RoboDK station: Simulare licenta.rdk

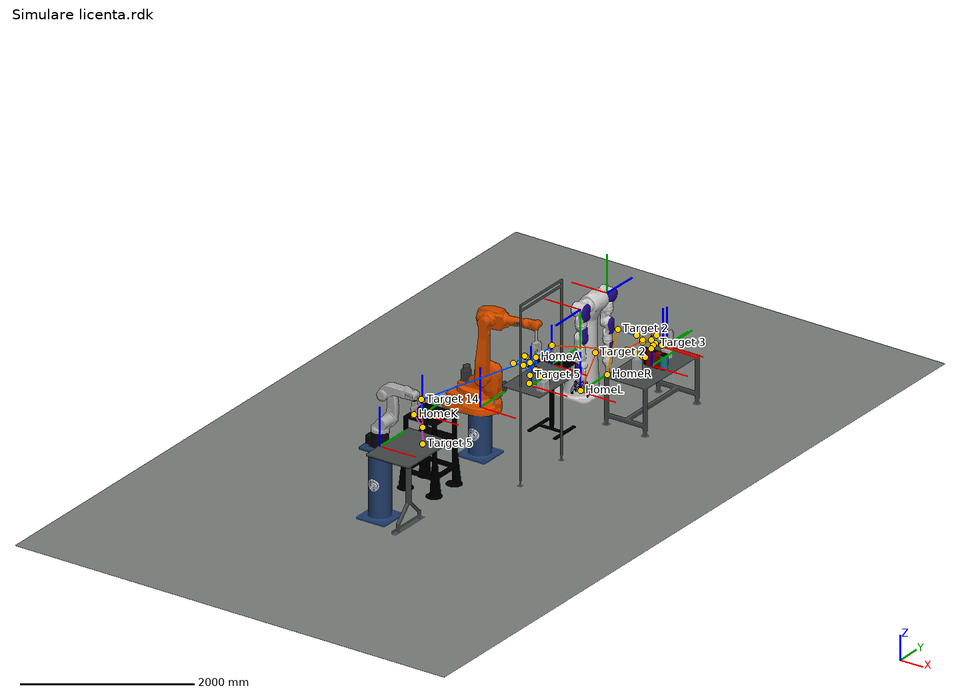
[picture v0: the station drawn from its stored meshes, robots at their saved joint values, targets as dots, program paths as lines]
Station Simulare licenta (saved by RoboDK 5.4.0). Poses are relative to the parent item; angles as X-Y-Z fixed-axis rotations.
  - frame ABB IRB 1600-6/1.45 Base at (0, 0, 600) mm
    - robot ABB IRB 1600-6/1.45: 6 axes, payload 6 kg, reach 1450 mm, repeatability 0.05 mm, weight 250 kg
        modified DH rows (alpha deg, a mm, theta deg, d mm): 0, 0, 0, 486.5; -90, 150, -90, 0; 0, 700, 0, 0; -90, 0, 0, 600; 90, 0, 0, 0; -90, 0, 180, 65
        joint limits [-180, -90, -245, -200, -115, -400] to [180, 120, 65, 200, 115, 400]; home [0, 0, 0, 0, 0, 0]; saved at [3.661, 0.324, -5.471, 0, 95.147, 3.661]
      - tool SCHUNK_0371103_PGN_plus_125_1__000, TCP at (0, 0, 350) mm, size 60 x 151.3 x 378 mm, geometry from SCHUNK_0371103_PGN_plus_125_1__000.stp
    - target HomeA (Cartesian target) at (750, 47.99, 825.32) mm, rotated rx 180 ry 0 rz -180 deg; joints [3.661, 0.324, -5.471, 0, 95.147, 3.661] of ABB IRB 1600-6/1.45
    - target Target 2 (Cartesian target) at (287.69, 1007.38, 456.93) mm, rotated rx 180 ry 0 rz -180 deg; joints [74.062, 29.214, -7.135, 0, 67.921, 74.062] of ABB IRB 1600-6/1.45
    - target Target 3 (Cartesian target) at (287.69, 1001.26, 332.84) mm, rotated rx 180 ry 0 rz -180 deg; joints [73.969, 33.457, -0.924, 0, 57.468, 73.969] of ABB IRB 1600-6/1.45
    - target Target 4 (Cartesian target) at (750, 47.99, 674.68) mm, rotated rx 180 ry 0 rz -180 deg; joints [3.661, 0.768, 8.512, 0, 80.72, 3.661] of ABB IRB 1600-6/1.45
    - target Target 5 (Cartesian target) at (852.72, -221.7, 732.38) mm, rotated rx 180 ry 89.49 rz 180 deg; joints [-26.861, -4.787, 53.092, 145.616, 53.133, -157.935] of ABB IRB 1600-6/1.45
    - target Target 6 (Cartesian target) at (849.34, -221.7, 627.88) mm, rotated rx 180 ry 89.49 rz 180 deg; joints [-27.04, 7.763, 58.334, 150.719, 68.35, -168.569] of ABB IRB 1600-6/1.45
    - target Target 7 (Cartesian target) at (750, -199.45, 825.32) mm, rotated rx 180 ry 0 rz -180 deg; joints [-14.893, 2.337, -7.538, 0, 95.202, -14.893] of ABB IRB 1600-6/1.45
    - target Target 8 (Cartesian target) at (854.13, -221.7, 892.62) mm, rotated rx 180 ry 89.5 rz 180 deg; joints [-26.786, -16.432, 42.285, 130.237, 36.18, -136.606] of ABB IRB 1600-6/1.45
    - target Target 9 (Cartesian target) at (925.55, -221.7, 818.94) mm, rotated rx 180 ry 44.11 rz -180 deg; joints [-19.198, -5.919, 12.219, 19.634, 42.934, -28.675] of ABB IRB 1600-6/1.45
    - target Target 10 (Cartesian target) at (925.55, -221.7, 818.94) mm, rotated rx 180 ry 89.61 rz 180 deg; joints [-23.472, -5.96, 42.941, 143.905, 42.537, -151.925] of ABB IRB 1600-6/1.45
    - target Target 11 (Cartesian target) at (623.92, -221.7, 821.01) mm, rotated rx 180 ry 89.61 rz 180 deg; joints [-46.699, -34.358, 57.99, 110.262, 50.873, -120.743] of ABB IRB 1600-6/1.45
    - target Target 12 (Cartesian target) at (636.73, 6.14, 820.92) mm, rotated rx -90.46 ry 31.14 rz -90.24 deg; joints [1.585, -46.941, 60.499, 6.927, -13.259, -65.588] of ABB IRB 1600-6/1.45
    - target Target 13 (Cartesian target) at (623.92, 5.25, 821.01) mm, rotated rx 180 ry 89.61 rz 180 deg; joints [1.44, -49.033, 60.724, 7.313, -11.39, -7.161] of ABB IRB 1600-6/1.45
    - target Target 14 (Cartesian target) at (-10.54, -1146, 546.53) mm, rotated rx 180 ry 0 rz -180 deg; joints [-90.527, 35.239, -25.964, -180, -80.725, 89.473] of ABB IRB 1600-6/1.45
    - target Target 15 (Cartesian target) at (-10.54, -1146, 387.82) mm, rotated rx 180 ry 0 rz -180 deg; joints [-90.527, 39.032, -16.756, -180, -67.724, 89.473] of ABB IRB 1600-6/1.45
    - target Target 16 (Cartesian target) at (287.69, 1019.67, 456.93) mm, rotated rx 180 ry 0 rz -180 deg; joints [74.244, 30.121, -8.606, 0, 68.485, 74.244] of ABB IRB 1600-6/1.45
    - target Target 17 (Cartesian target) at (985.75, -221.7, 756.85) mm, rotated rx 180 ry 44.11 rz -180 deg; joints [-17.647, -0.333, 13.009, 20.817, 36.422, -29.877] of ABB IRB 1600-6/1.45
    - target Target 18 (Cartesian target) at (985.75, -221.7, 756.85) mm, rotated rx 180 ry 89.15 rz 180 deg; joints [-21.226, 2.977, 41.791, 150.728, 47.764, -159.685] of ABB IRB 1600-6/1.45
    - target Target 19 (Cartesian target) at (985.75, -221.7, 756.85) mm, rotated rx 180 ry 44.11 rz -180 deg; joints [-17.647, -0.333, 13.009, 20.817, 36.422, -29.877] of ABB IRB 1600-6/1.45
    - target Target 20 (Cartesian target) at (985.75, -221.7, 756.85) mm, rotated rx 180 ry 89.15 rz 180 deg; joints [-21.226, 2.977, 41.791, 150.728, 47.764, -159.685] of ABB IRB 1600-6/1.45
  - frame KUKA KR 5 sixx R850 Base at (0, -2000, 900) mm
    - robot KUKA KR 5 sixx R850: 6 axes, payload 5 kg, reach 855 mm, repeatability 0.03 mm, weight 29 kg
        modified DH rows (alpha deg, a mm, theta deg, d mm): 0, 0, 0, 335; -90, 75, 0, 0; 0, 365, -90, 0; -90, 90, 0, 405; 90, 0, 0, 0; -90, 0, 180, 80
        joint limits [-170, -190, -119, -190, -120, -358] to [170, 45, 165, 190, 120, 358]; home [0, -90, 90, 0, 0, 0]; saved at [0, -90, 90, 0, 90, 0]
      - tool 539635_HGP_25_A_B_SSK____asm_0__ZH_, TCP at (0, 0, 170) mm, rotated rx 0 ry 0 rz 180 deg, size 47 x 101 x 197.2 mm, geometry from 539635_HGP_25_A_B_SSK____asm_0__ZH_.stp
    - target HomeK (Cartesian target) at (480, 0, 540) mm, rotated rx -180 ry 0 rz 0 deg; joints [0, -90, 90, 0, 90, 0] of KUKA KR 5 sixx R850
    - target Target 2 (Cartesian target) at (-12.02, 851.6, 253.67) mm, rotated rx 92.47 ry -89.16 rz 180 deg; joints [-90.12, -42.173, 106.544, 2.603, -64.358, -0.286] of KUKA KR 5 sixx R850
    - target Target 4 (Cartesian target) at (577.64, 29.88, 390.74) mm, rotated rx 1.04 ry -89.16 rz 180 deg; joints [-4.42, -93.031, 154.413, -3.815, -62.276, 1.842] of KUKA KR 5 sixx R850
    - target Target 5 (Cartesian target) at (579.54, 29.86, 183.27) mm, rotated rx 1.04 ry -89.16 rz 180 deg; joints [-4.391, -45.31, 147.993, -3.443, -103.501, -0.74] of KUKA KR 5 sixx R850
    - target Target 6 (Cartesian target) at (480, 0, 540) mm, rotated rx -180 ry 0 rz 0 deg; joints [0, -90, 90, 0, 90, 0] of KUKA KR 5 sixx R850
    - target Target 7 (Cartesian target) at (-12.02, 851.6, 253.67) mm, rotated rx 92.47 ry -89.16 rz 180 deg; joints [-90.12, -42.173, 106.544, 2.603, -64.358, -0.286] of KUKA KR 5 sixx R850
    - target Target 7 (Cartesian target) at (-9.43, 851.6, 77.3) mm, rotated rx 92.47 ry -89.16 rz 180 deg; joints [-89.873, -18.515, 95.22, 2.665, -76.682, 0.227] of KUKA KR 5 sixx R850
  - object Pedestal H36in at (0, 0, 0) mm, size 400 x 400 x 914.4 mm, geometry from Pedestal-H36in.sld
  - object masaabb at (0, 0, 0) mm, size 880 x 530 x 2305 mm, geometry from masaabb.stp
  - object Pedestal H24in at (0, 0, 0) mm, size 400 x 400 x 609.6 mm, geometry from Pedestal-H24in.sld
  - object masakuka at (0, 0, 0) mm, size 600 x 850 x 1000 mm, geometry from masakuka.stp
  - object masaintreroboti at (0, -1000, 0) mm, size 600 x 600 x 910 mm, geometry from masaintreroboti.stp
  - frame Frame 6 at (1000, 2000, 610) mm, rotated rx 0.04 ry 0 rz 0 deg
    - object masamotoman at (0, 0, 0) mm, size 640 x 1140 x 615 mm, geometry from masamotoman.stp
    - object suport pahare at (0, -300, 0) mm, rotated rx 0 ry 0 rz 180 deg, size 100 x 100 x 210 mm, geometry from suport pahare.stp
    - object Suport cafea at (0, 0, 0) mm, size 151.2 x 153.3 x 313 mm, geometry from Suport cafea.stl
  - frame Motoman CSDA10F Base at (0, 2000, 0) mm
    - robot Turntable: 1 axes
        modified DH rows (alpha deg, a mm, theta deg, d mm): 0, 0, 0, 0
        base shift (92.5, 0, 0) mm
        joint limits [-200] to [200]; home [0]; saved at [0]
      - frame Right Arm at (100, 265, 1200) mm, rotated rx 90 ry 0 rz -180 deg
        - robot Right CSDA10F (model Motoman CSDA10F): 7 axes, payload 10 kg, reach 720 mm, repeatability 0.6 mm, weight 60 kg
            modified DH rows (alpha deg, a mm, theta deg, d mm): 0, 0, 0, 360; -90, 0, 0, 0; 90, 0, 0, 360; -90, 0, 0, 0; 90, 0, 0, 360; -90, 0, 0, 0; 90, 0, 180, 175
            base shift (0, 0, -360) mm
            joint limits [-180, -110, -170, -135, -180, -110, -180] to [180, 110, 170, 135, 180, 110, 180]; home [90, -90, -90, -130, 0, -60, 90]; saved at [90, -90, 0, 0, 0, 0, 0]
          - tool LEHZ20K2_10_16_0_, TCP at (0, 0, 140) mm, size 81.3 x 34.5 x 159.6 mm, geometry from LEHZ20K2_10_16_0_.stp
        - target HomeR (Cartesian target) at (0, -1035, 0) mm, rotated rx 0 ry 90 rz -90 deg; joints [90, -90, 0, 0, 0, 0, 0] of Right CSDA10F
        - target Target 2 (Cartesian target) at (-146.78, -414.63, 0) mm, rotated rx 0 ry 90 rz -179.5 deg; joints [112.215, -38.164, 0, -103.672, 107.385, 103.215, -36.135] of Right CSDA10F
        - target Target 3 (Cartesian target) at (-649.29, -465.08, 33.19) mm, rotated rx 0 ry 90 rz -179.5 deg; joints [54.13, -49.207, 0, -74.927, 67.545, 60.603, -49.904] of Right CSDA10F
        - target Target 4 (Cartesian target) at (-742.98, -465.91, 33.19) mm, rotated rx 0 ry 90 rz -179.5 deg; joints [47.259, -58.279, 0, -57.417, 67.815, 51.877, -56.553] of Right CSDA10F
        - target Target 5 (Cartesian target) at (-679.15, -330.72, -257.56) mm, rotated rx 0 ry 90 rz -179.5 deg; joints [42.006, -77.982, 0, -79.484, 43.77, 73.322, -15.373] of Right CSDA10F
        - target Target 6 (Cartesian target) at (-821.86, -332.03, -257.56) mm, rotated rx 0 ry 90 rz -179.5 deg; joints [33.009, -88.937, 0, -48.286, 40.963, 55.058, -26.438] of Right CSDA10F
        - target Target 7 (Cartesian target) at (-602.81, -256.65, -278.95) mm, rotated rx 0 ry 90 rz -179.5 deg; joints [41.415, -77.232, 0, -97.556, 41.03, 86.064, -3.419] of Right CSDA10F
        - target Target 8 (Cartesian target) at (-813.1, -258.6, -278.95) mm, rotated rx 0 ry 90 rz -179.5 deg; joints [27.186, -86.811, 0, -59.339, 31.181, 60.152, -16.762] of Right CSDA10F
        - target Target 9 (Cartesian target) at (-812.16, -365.94, -278.95) mm, rotated rx 0 ry 90 rz -179.5 deg; joints [36.148, -94.225, 0, -40.297, 45.644, 54.592, -30.649] of Right CSDA10F
        - target Target 10 (Cartesian target) at (-538.22, -468.56, 212.74) mm, rotated rx -180 ry 62.97 rz 0.5 deg; joints [61.069, -29.073, 0, -54.35, 122.881, 67.492, -110.522] of Right CSDA10F
        - target Target 11 (Cartesian target) at (-766.53, -470.56, 96.28) mm, rotated rx 180 ry 62.97 rz 0.5 deg; joints [43.929, -64.378, 0, -12.171, 134.051, 58.432, -128.308] of Right CSDA10F
      - frame Left Arm at (100, -265, 1200) mm, rotated rx -90 ry 0 rz 180 deg
        - robot Left CSDA10F (model Motoman CSDA10F): 7 axes, payload 10 kg, reach 720 mm, repeatability 0.6 mm, weight 60 kg
            modified DH rows (alpha deg, a mm, theta deg, d mm): 0, 0, 0, 360; -90, 0, 0, 0; 90, 0, 0, 360; -90, 0, 0, 0; 90, 0, 0, 360; -90, 0, 0, 0; 90, 0, 180, 175
            base shift (0, 0, -360) mm
            joint limits [-180, -110, -170, -135, -180, -110, -180] to [180, 110, 170, 135, 180, 110, 180]; home [90, 90, -90, -130, 0, -60, 90]; saved at [-90.45, -90.93, 0, 0, 90, 0, -90]
          - tool ROBOTIQ_AGS-001-XXXX_20171116, TCP at (0, 0, 150) mm, size 130.2 x 233.3 x 211.5 mm, geometry from ROBOTIQ_AGS-001-XXXX_20171116.STEP
        - target Target 2 (Cartesian target) at (-208.84, 486.87, 0) mm, rotated rx -90 ry -0.83 rz 89.91 deg; joints [-102.313, -43.74, 0, -92.52, -98.892, 98.414, -47.744] of Left CSDA10F
        - target Target 3 (Cartesian target) at (-669.86, 304.45, 44.19) mm, rotated rx -90 ry -0.83 rz 89.91 deg; joints [-40.579, -35.277, 0, -98.641, -50.903, 56.779, -56.839] of Left CSDA10F
        - target Target 8 (Cartesian target) at (-669.91, 304.4, 43.85) mm, rotated rx 90 ry 0.78 rz -90.09 deg; joints [-40.571, -35.314, 0, -98.646, -50.877, 56.802, 123.169] of Left CSDA10F
        - target Target 5 (Cartesian target) at (-669.9, 307.55, -277.75) mm, rotated rx 90 ry 0.78 rz -90.09 deg; joints [-40.865, -79.854, 0, -81.531, -42.301, 76.009, 101.628] of Left CSDA10F
        - target Target 6 (Cartesian target) at (-669.56, 518.22, -278.86) mm, rotated rx 90 ry 0.78 rz -90.09 deg; joints [-55.594, -96.456, 0, -35.009, -65.533, 64.885, 132.227] of Left CSDA10F
        - target Target 7 (Cartesian target) at (-705.87, 518.26, -277) mm, rotated rx 90 ry 0.78 rz -90.09 deg; joints [-52.949, -101.558, 0, -23.127, -66.682, 60.23, 138.259] of Left CSDA10F
        - target Target 9 (Cartesian target) at (-100.6, 140.55, 710.33) mm, rotated rx 0.4 ry 0.69 rz -90.09 deg; joints [-55.715, 29.267, 0, -106.213, -0.736, 77.293, 145.784] of Left CSDA10F
        - target Target 10 (Cartesian target) at (-110.24, 293.24, 712.34) mm, rotated rx 0.4 ry 0.78 rz -90.09 deg; joints [-70.041, 6.583, 0, -90.245, -0.643, 84.256, 160.014] of Left CSDA10F
        - target Target 11 (Cartesian target) at (-669.91, 304.4, 43.85) mm, rotated rx 90 ry 0.78 rz -90.09 deg; joints [-40.571, -35.314, 0, -98.646, -50.877, 56.802, 123.169] of Left CSDA10F
        - target Target 12 (Cartesian target) at (-785.67, 306.43, 46.88) mm, rotated rx -90 ry 0 rz 90.02 deg; joints [-33.642, -45.628, 0, -79.058, -49.489, 46.813, -51.306] of Left CSDA10F
        - target Target 12 (Cartesian target) at (-785.67, 306.43, 46.88) mm, rotated rx -90 ry 0 rz 90.02 deg; joints [-33.077, -46.752, 0, -76.954, -49.594, 45.821, -50.694] of Left CSDA10F
        - target HomeL (Cartesian target) at (8.13, 1034.83, -16.8) mm, rotated rx -180 ry 89.07 rz -90.45 deg; joints [-90.45, -90.93, 0, 0, 90, 0, -90] of Left CSDA10F
  - program Capula neagra (18 instructions, listed below)
  - program Prog2 (21 instructions, listed below)
  - program Program Motoman (2 instructions, listed below)
  - object masaintremotoabb at (0, 0, 0) mm, size 400 x 400 x 860 mm, geometry from masaintremotoabb.stp
  - program Prog4 (39 instructions, listed below)
  - program Prog5 (12 instructions, listed below)
  - program Prog6 (5 instructions, listed below)
  - frame Frame 7 at (1000, 2000, 610) mm
    - object Nesspreso Essensa Mini v11 at (0, 0, 0) mm, size 330.3 x 112.6 x 205.3 mm, geometry from Nesspreso Essensa Mini v11.iges
  - program Prog7 (6 instructions, listed below)
  - frame Frame 8 at (300, 1000, 830) mm
  - frame Frame 9 at (0, -1145.9, 968.34) mm
    - target Target 3 (Cartesian target) at (-9.43, -2.5, 8.97) mm, rotated rx 92.47 ry -89.16 rz 180 deg; joints [-89.873, -18.515, 95.22, 2.665, -76.682, 0.227] of KUKA KR 5 sixx R850
  - frame Frame 10 at (950, 2300.45, 710) mm
    - object Dolce Gusto capsule at (0, 0, 0) mm, size 53.2 x 54 x 34.7 mm, geometry from Dolce Gusto capsule.STEP
  - frame Frame 11 at (870, -220, 1206) mm
    - object recipient zahar at (160.01, 0.07, -5.93) mm, rotated rx -0.02 ry -0.02 rz 90.02 deg, size 123.8 x 125.4 x 140.2 mm, geometry from recipient zahar.stp
    - object lingurita at (0, 0, 0) mm, size 99.2 x 40.9 x 19 mm, geometry from lingurita.stp
  - object podea at (0, 0, -3) mm, rotated rx 0 ry 0 rz 90 deg, size 10000 x 6000 x 2 mm, geometry from podea.stp
  - Python program mqtt_joints_motoman_left (listed below)
  - Python program mqtt_joints_motoman_right (listed below)
  - Python program mqtt_joints_kuka (listed below)
  - Python program mqtt_joints_abb (listed below)
  - Python program cafea (listed below)
  - program Capsula lapte (19 instructions, listed below)
  - frame Frame 12 at (970, 2350.45, 710) mm
    - object Dolce Gusto capsule at (0, 0, 0) mm, size 53.2 x 54 x 34.7 mm, geometry from Dolce Gusto capsule.STEP
  - program 2 lingurite (47 instructions, listed below)
  - program 3 lingurite (55 instructions, listed below)
  - program neagra2 (6 instructions, listed below)
  - program neagra3 (6 instructions, listed below)
  - program lapte1 (6 instructions, listed below)
  - program lapte2 (6 instructions, listed below)
  - program lapte3 (6 instructions, listed below)
  - object Coffee Cup- at (1000, 1700, 900) mm, size 84.6 x 83.8 x 116.5 mm, geometry from Coffee Cup-.STEP
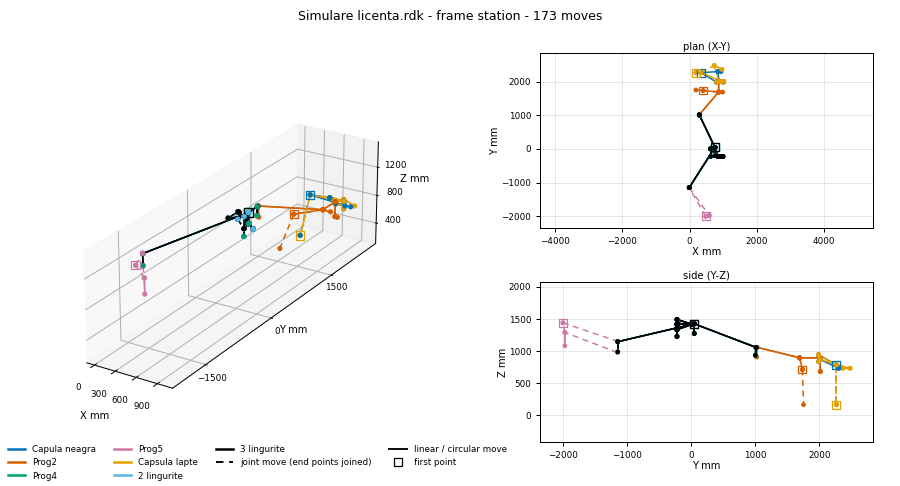
[picture p0: tool path of Simulare licenta.rdk in frame station, 173 of 173 moves have a stored position in this frame; points joined in program order, loops and branches not executed]

--- program Capula neagra (robot Right CSDA10F) ---
  Set Ref.: Right Arm
  MoveJ (Target 2)
  MoveL (Target 3)
  MoveL (Target 4)
  Attach to LEHZ20K2_10_16_0_
  MoveL (Target 3)
  MoveL (Target 5)
  MoveL (Target 6)
  Detach from LEHZ20K2_10_16_0_
  Hide Dolce Gusto capsule
  MoveL (Target 5)
  MoveL (Target 7)
  MoveL (Target 8)
  MoveL (Target 9)
  MoveL (Target 8)
  MoveL (Target 7)
  MoveL (Target 2)
  MoveJ (HomeR)

--- program Prog2 (robot Left CSDA10F) ---
  Set Ref.: Left Arm
  MoveJ (Target 2)
  MoveL (Target 3)
  MoveL (Target 12)
  Attach to ROBOTIQ_AGS-001-XXXX_20171116
  MoveL (Target 3)
  MoveJ (Target 8)
  MoveL (Target 5)
  MoveL (Target 6)
  MoveL (Target 7)
  Pause 10.0 s
  MoveL (Target 6)
  MoveL (Target 5)
  MoveL (Target 8)
  MoveL (Target 9)
  MoveL (Target 10)
  Detach from ROBOTIQ_AGS-001-XXXX_20171116
  MoveL (Target 9)
  MoveL (Target 11)
  MoveJ (Target 2)
  MoveJ (Target 13) -> target HomeL

--- program Program Motoman (robot ABB IRB 1600-6/1.45) ---
  Call Capula neagra
  Call Prog2

--- program Prog4 (robot ABB IRB 1600-6/1.45) ---
  Set Ref.: ABB IRB 1600-6/1.45 Base
  MoveJ (HomeA)
  MoveL (Target 16)
  MoveL (Target 3)
  Attach to SCHUNK_0371103_PGN_plus_125_1__000
  MoveL (Target 2)
  MoveL (HomeA)
  MoveL (Target 4)
  Detach from SCHUNK_0371103_PGN_plus_125_1__000
  MoveL (HomeA)
  MoveL (Target 7)
  MoveJ (Target 5)
  MoveL (Target 6)
  Attach to SCHUNK_0371103_PGN_plus_125_1__000
  MoveL (Target 5)
  MoveL (Target 10)
  MoveJ (Target 9)
  MoveL (Target 19)
  MoveL (Target 20)
  MoveL (Target 10)
  MoveL (Target 8)
  MoveL (Target 13)
  MoveJ (Target 12)
  MoveJ (Target 13)
  MoveL (Target 11)
  MoveL (Target 8)
  MoveL (Target 5)
  MoveL (Target 6)
  Detach from SCHUNK_0371103_PGN_plus_125_1__000
  MoveL (Target 5)
  MoveL (HomeA)
  MoveL (Target 4)
  Attach to SCHUNK_0371103_PGN_plus_125_1__000
  MoveL (HomeA)
  MoveL (Target 14)
  MoveL (Target 15)
  Detach from SCHUNK_0371103_PGN_plus_125_1__000
  MoveL (Target 14)
  MoveL (HomeA)

--- program Prog5 (robot KUKA KR 5 sixx R850) ---
  Set Ref.: KUKA KR 5 sixx R850 Base
  Set Tool: 539635_HGP_25_A_B_SSK____asm_0__ZH_
  MoveJ (Target 6)
  MoveJ (Target 7)
  MoveL (Target 2)
  MoveL (Target 7)
  Attach to 539635_HGP_25_A_B_SSK____asm_0__ZH_
  MoveJ (Target 4)
  MoveL (Target 5)
  Detach from 539635_HGP_25_A_B_SSK____asm_0__ZH_
  MoveL (Target 4)
  MoveJ (HomeK)

--- program Prog6 (robot ABB IRB 1600-6/1.45) ---
  Call Program Motoman
  Call Prog4
  Call Prog5
  Pause 5.0 s
  Call Prog7

--- program Prog7 (robot ABB IRB 1600-6/1.45) ---
  Replace objects
  Replace objects
  Show Dolce Gusto capsule
  Replace objects
  Replace Dolce Gusto capsule
  Show Dolce Gusto capsule

--- Python program mqtt_joints_motoman_left ---
import random

from paho.mqtt import client as mqtt_client

from robodk.robolink import *

RDK = Robolink()
robot  = RDK.Item('Left CSDA10F')

broker = '188.24.48.213'
#broker = '192.168.1.113'
port = 1883
topic = "licenta/jointsmotomanl"
# generate client ID with pub prefix randomly
client_id = f'python-mqtt-{random.randint(0, 100)}'
username = 'basti'
password = 'topsecret'


def connect_mqtt() -> mqtt_client:
    def on_connect(client, userdata, flags, rc):
        if rc == 0:
            print("Connected to MQTT Broker!")
        else:
            print("Failed to connect, return code %d\n", rc)

    client = mqtt_client.Client(client_id)
    client.username_pw_set(username, password)
    client.on_connect = on_connect
    client.connect(broker, port)
    return client

def filtrare (mesaj):
    nc = "{},:'jml "
    for character in nc:
        mesaj = mesaj.replace(character, "")
    j = mesaj.split('"')
    indices = [2, 4, 6, 8, 10, 12, 14]
    print(mesaj)
    extracted_elements = [j[index] for index in indices]
    for i in range(0, len(extracted_elements)):
        extracted_elements[i] = int(extracted_elements[i])
    return extracted_elements

def subscribe(client: mqtt_client):
    def on_message(client, userdata, msg):
        mesaj = msg.payload.decode()
        joints = filtrare(mesaj)
        robot.MoveJ(joints)
    client.subscribe(topic)
    client.on_message = on_message


def run():
    client = connect_mqtt()
    subscribe(client)
    client.loop_forever()


if __name__ == '__main__':
    run()

--- Python program mqtt_joints_motoman_right ---
import random

from paho.mqtt import client as mqtt_client

from robodk.robolink import *

RDK = Robolink()
robot  = RDK.Item('Right CSDA10F')

broker = '188.24.48.213'
#broker = '192.168.1.113'
port = 1883
topic = "licenta/jointsmotomanr"
# generate client ID with pub prefix randomly
client_id = f'python-mqtt-{random.randint(0, 100)}'
username = 'basti'
password = 'topsecret'


def connect_mqtt() -> mqtt_client:
    def on_connect(client, userdata, flags, rc):
        if rc == 0:
            print("Connected to MQTT Broker!")
        else:
            print("Failed to connect, return code %d\n", rc)

    client = mqtt_client.Client(client_id)
    client.username_pw_set(username, password)
    client.on_connect = on_connect
    client.connect(broker, port)
    return client


def filtrare (mesaj):
    nc = "{},:'jmr "
    for character in nc:
        mesaj = mesaj.replace(character, "")
    j = mesaj.split('"')
    indices = [2, 4, 6, 8, 10, 12, 14]
    print(mesaj)
    extracted_elements = [j[index] for index in indices]
    for i in range(0, len(extracted_elements)):
        extracted_elements[i] = int(extracted_elements[i])
    return extracted_elements

def subscribe(client: mqtt_client):
    def on_message(client, userdata, msg):
        mesaj = msg.payload.decode()
        joints = filtrare(mesaj)
        robot.MoveJ(joints)
    client.subscribe(topic)
    client.on_message = on_message


def run():
    client = connect_mqtt()
    subscribe(client)
    client.loop_forever()


if __name__ == '__main__':
    run()

--- Python program mqtt_joints_kuka ---
import random

from paho.mqtt import client as mqtt_client

from robodk.robolink import *

#broker = '192.168.1.113'
broker = '188.24.48.213'
port = 1883
topic = "licenta/jointskuka"
client_id = f'python-mqtt-{random.randint(0, 100)}'
username = 'basti'
password = 'topsecret'
RDK = Robolink()
robot  = RDK.Item('KUKA KR 5 sixx R850')

def connect_mqtt() -> mqtt_client:
    def on_connect(client, userdata, flags, rc):
        if rc == 0:
            print("Connected to MQTT Broker!")
        else:
            print("Failed to connect, return code %d\n", rc)

    client = mqtt_client.Client(client_id)
    client.username_pw_set(username, password)
    client.on_connect = on_connect
    client.connect(broker, port)
    return client


def filtrare(mesaj):
    nc = "{},:'jk "
    for character in nc:
            mesaj = mesaj.replace(character, "")
    j = mesaj.split('"')
    indices = [2, 4, 6, 8, 10, 12]
    print(mesaj)
    extracted_elements = [j[index] for index in indices]
    for i in range(0, len(extracted_elements)):
        extracted_elements[i] = int(extracted_elements[i])
    return extracted_elements

def subscribe(client: mqtt_client):
    def on_message(client, userdata, msg):
        mesaj = msg.payload.decode()
        joints = filtrare(mesaj)
        robot.MoveJ(joints)
    client.subscribe(topic)
    client.on_message = on_message


def run():
    client = connect_mqtt()
    subscribe(client)
    client.loop_forever()


if __name__ == '__main__':
    run()

--- Python program mqtt_joints_abb ---
import random

from paho.mqtt import client as mqtt_client

from robodk.robolink import *

RDK = Robolink()
robot  = RDK.Item('ABB IRB 1600-6/1.45')

broker = '188.24.48.213'
#broker = '192.168.1.113'
port = 1883
topic = "licenta/jointsabb"
# generate client ID with pub prefix randomly
client_id = f'python-mqtt-{random.randint(0, 100)}'
username = 'basti'
password = 'topsecret'


def connect_mqtt() -> mqtt_client:
    def on_connect(client, userdata, flags, rc):
        if rc == 0:
            print("Connected to MQTT Broker!")
        else:
            print("Failed to connect, return code %d\n", rc)

    client = mqtt_client.Client(client_id)
    client.username_pw_set(username, password)
    client.on_connect = on_connect
    client.connect(broker, port)
    return client


def filtrare (mesaj):
    nc = "{},:'ja "
    for character in nc:
        mesaj = mesaj.replace(character, "")
    j = mesaj.split('"')
    indices = [2, 4, 6, 8, 10, 12]
    print(mesaj)
    extracted_elements = [j[index] for index in indices]
    for i in range(0, len(extracted_elements)):
        extracted_elements[i] = int(extracted_elements[i])
    return extracted_elements

def subscribe(client: mqtt_client):
    def on_message(client, userdata, msg):
        mesaj = msg.payload.decode()
        joints = filtrare(mesaj)
        robot.MoveJ(joints)
    client.subscribe(topic)
    client.on_message = on_message


def run():
    client = connect_mqtt()
    subscribe(client)
    client.loop_forever()


if __name__ == '__main__':
    run()

--- Python program cafea ---
import random

from paho.mqtt import client as mqtt_client

from robodk.robolink import *

RDK = Robolink()
robot  = RDK.Item('ABB IRB 1600-6/1.45')
case1 = RDK.Item('Prog6')
case2 = RDK.Item('neagra2')
case3 = RDK.Item('neagra3')
case4 = RDK.Item('lapte1')
case5 = RDK.Item('lapte2')
case6 = RDK.Item('lapte3')

broker = '188.24.48.213'
#broker = '192.168.1.113'
port = 1883
topic = "licenta/cafea"
# generate client ID with pub prefix randomly
client_id = f'python-mqtt-{random.randint(0, 100)}'
username = 'basti'
password = 'topsecret'


def connect_mqtt() -> mqtt_client:
    def on_connect(client, userdata, flags, rc):
        if rc == 0:
            print("Connected to MQTT Broker!")
        else:
            print("Failed to connect, return code %d\n", rc)

    client = mqtt_client.Client(client_id)
    client.username_pw_set(username, password)
    client.on_connect = on_connect
    client.connect(broker, port)
    return client


def caseSelection (mesaj):
    case = int(mesaj)
    print(case)
    if case == 21:
        case1.RunProgram()
        while case1.Busy():
            print("Waiting for the program to complete")
    elif case == 25:
        case2.RunProgram()
        while case2.Busy():
            print("Waiting for the program to complete")
    elif case == 27:
        case3.RunProgram()
        while case3.Busy():
            print("Waiting for the program to complete")
    elif case == 31:
        case4.RunProgram()
        while case4.Busy():
            print("Waiting for the program to complete")
    elif case == 35:
        case5.RunProgram()
        while case5.Busy():
            print("Waiting for the program to complete")
    elif case == 37:
        case6.RunProgram()
        while case6.Busy():
            print("Waiting for the program to complete")

def subscribe(client: mqtt_client):
    def on_message(client, userdata, msg):
        mesaj = msg.payload.decode()
        caseSelection(mesaj)
    client.subscribe(topic)
    client.on_message = on_message


def run():
    client = connect_mqtt()
    subscribe(client)
    client.loop_forever()


if __name__ == '__main__':
    run()

--- program Capsula lapte (robot Right CSDA10F) ---
  Set Ref.: Right Arm
  Set Tool: LEHZ20K2_10_16_0_
  MoveJ (HomeR)
  MoveJ (Target 2)
  MoveJ (Target 10)
  MoveL (Target 11)
  Attach to LEHZ20K2_10_16_0_
  MoveL (Target 10)
  MoveL (Target 5)
  MoveL (Target 6)
  Detach from LEHZ20K2_10_16_0_
  Hide Dolce Gusto capsule
  MoveL (Target 5)
  MoveL (Target 7)
  MoveL (Target 8)
  MoveL (Target 9)
  MoveL (Target 8)
  MoveL (Target 2)
  MoveJ (HomeR)

--- program 2 lingurite (robot ABB IRB 1600-6/1.45) ---
  Set Ref.: ABB IRB 1600-6/1.45 Base
  MoveJ (HomeA)
  MoveL (Target 16)
  MoveL (Target 3)
  Attach to SCHUNK_0371103_PGN_plus_125_1__000
  MoveL (Target 2)
  MoveL (HomeA)
  MoveL (Target 4)
  Detach from SCHUNK_0371103_PGN_plus_125_1__000
  MoveL (HomeA)
  MoveL (Target 7)
  MoveJ (Target 5)
  MoveL (Target 6)
  Attach to SCHUNK_0371103_PGN_plus_125_1__000
  MoveL (Target 5)
  MoveL (Target 10)
  MoveJ (Target 9)
  MoveL (Target 19)
  MoveL (Target 20)
  MoveL (Target 10)
  MoveL (Target 8)
  MoveL (Target 13)
  MoveJ (Target 12)
  MoveJ (Target 13)
  MoveJ (Target 9)
  MoveL (Target 19)
  MoveL (Target 20)
  MoveL (Target 10)
  MoveL (Target 8)
  MoveL (Target 13)
  MoveJ (Target 12)
  MoveJ (Target 13)
  MoveL (Target 11)
  MoveL (Target 8)
  MoveL (Target 5)
  MoveL (Target 6)
  Detach from SCHUNK_0371103_PGN_plus_125_1__000
  MoveL (Target 5)
  MoveL (HomeA)
  MoveL (Target 4)
  Attach to SCHUNK_0371103_PGN_plus_125_1__000
  MoveL (HomeA)
  MoveL (Target 14)
  MoveL (Target 15)
  Detach from SCHUNK_0371103_PGN_plus_125_1__000
  MoveL (Target 14)
  MoveL (HomeA)

--- program 3 lingurite (robot ABB IRB 1600-6/1.45) ---
  Set Ref.: ABB IRB 1600-6/1.45 Base
  MoveJ (HomeA)
  MoveL (Target 16)
  MoveL (Target 3)
  Attach to SCHUNK_0371103_PGN_plus_125_1__000
  MoveL (Target 2)
  MoveL (HomeA)
  MoveL (Target 4)
  Detach from SCHUNK_0371103_PGN_plus_125_1__000
  MoveL (HomeA)
  MoveL (Target 7)
  MoveJ (Target 5)
  MoveL (Target 6)
  Attach to SCHUNK_0371103_PGN_plus_125_1__000
  MoveL (Target 5)
  MoveL (Target 10)
  MoveJ (Target 9)
  MoveL (Target 19)
  MoveL (Target 20)
  MoveL (Target 10)
  MoveL (Target 8)
  MoveL (Target 13)
  MoveJ (Target 12)
  MoveJ (Target 13)
  MoveJ (Target 9)
  MoveL (Target 19)
  MoveL (Target 20)
  MoveL (Target 10)
  MoveL (Target 8)
  MoveL (Target 13)
  MoveJ (Target 12)
  MoveJ (Target 13)
  MoveJ (Target 9)
  MoveL (Target 19)
  MoveL (Target 20)
  MoveL (Target 10)
  MoveL (Target 8)
  MoveL (Target 13)
  MoveJ (Target 12)
  MoveJ (Target 13)
  MoveL (Target 11)
  MoveL (Target 8)
  MoveL (Target 5)
  MoveL (Target 6)
  Detach from SCHUNK_0371103_PGN_plus_125_1__000
  MoveL (Target 5)
  MoveL (HomeA)
  MoveL (Target 4)
  Attach to SCHUNK_0371103_PGN_plus_125_1__000
  MoveL (HomeA)
  MoveL (Target 14)
  MoveL (Target 15)
  Detach from SCHUNK_0371103_PGN_plus_125_1__000
  MoveL (Target 14)
  MoveL (HomeA)

--- program neagra2 (robot ABB IRB 1600-6/1.45) ---
  Call Capula neagra
  Call Prog2
  Call 2 lingurite
  Call Prog5
  Pause 5.0 s
  Call Prog7

--- program neagra3 (robot ABB IRB 1600-6/1.45) ---
  Call Capula neagra
  Call Prog2
  Call 3 lingurite
  Call Prog5
  Pause 5.0 s
  Call Prog7

--- program lapte1 (robot ABB IRB 1600-6/1.45) ---
  Call Capsula lapte
  Call Prog2
  Call Prog4
  Call Prog5
  Pause 5.0 s
  Call Prog7

--- program lapte2 (robot ABB IRB 1600-6/1.45) ---
  Call Capsula lapte
  Call Prog2
  Call 2 lingurite
  Call Prog5
  Pause 5.0 s
  Call Prog7

--- program lapte3 (robot ABB IRB 1600-6/1.45) ---
  Call Capsula lapte
  Call Prog2
  Call 3 lingurite
  Call Prog5
  Pause 5.0 s
  Call Prog7
